// TIA Portal V18 export
FUNCTION "myFunction" : Void   // FC1, LAD
{ S7_Optimized_Access := 'TRUE' }
VERSION : 0.1
// stored: AutoNumber true, IsIECCheckEnabled false, SetENOAutomatically false, UDAEnableTagReadback false
BEGIN

REGION Network 1
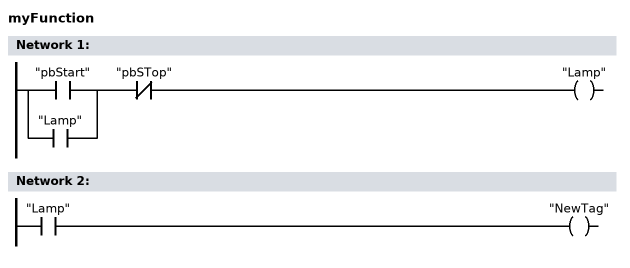
   RUNG wire#powerrail
      Contact( "pbStart" )
      wire#w1
      I_Contact( "pbSTop" )
      Coil( "Lamp" )
   END_RUNG
   RUNG wire#powerrail
      Contact( "Lamp" )
   END_RUNG wire#w1
   // the same network as SCL:
   "Lamp" := ("pbStart" OR "Lamp") AND NOT "pbSTop";
END_REGION

REGION Network 2
   RUNG wire#powerrail
      Contact( "Lamp" )
      Coil( "NewTag" )
   END_RUNG
   // the same network as SCL:
   "NewTag" := "Lamp";
END_REGION
END_FUNCTION
